{attribute 'enable_dynamic_creation'}
FUNCTION_BLOCK NotificationIterator IMPLEMENTS Iterator
VAR
	pNotificationList 	: ARRAY[0..Param.MAX_ITERABLE_ITEMS] OF POINTER TO Notification;
	//pNotification 		: POINTER TO Notification; 
	nPosition 			: INT := 0;
END_VAR

METHOD current : Object
VAR
	pNotification 		: POINTER TO Notification; 
END_VAR
pNotification := THIS^.pNotificationList[nPosition];
current := pNotification^;
END_METHOD

METHOD FB_init : BOOL
VAR_INPUT
	bInitRetains : BOOL; // if TRUE, the retain variables are initialized (warm start / cold start)
	bInCopyCode : BOOL;  // if TRUE, the instance afterwards gets moved into the copy code (online change)
	pNotificationList : ARRAY[0..Param.MAX_ITERABLE_ITEMS] OF POINTER TO Notification;
END_VAR
This^.pNotificationList := pNotificationList;
END_METHOD

METHOD hasNext : BOOL
IF (THIS^.pNotificationList[nPosition + 1] <> 16#0000) THEN
	hasNext := TRUE;
ELSE
	hasNext := FALSE;	
END_IF
END_METHOD

METHOD next : Object
VAR
	pNotification 		: POINTER TO Notification; 
END_VAR
THIS^.nPosition := THIS^.nPosition + 1;

pNotification := THIS^.pNotificationList[nPosition];
next := pNotification^;
END_METHOD

PROPERTY Position : INT
GET
Position := nPosition;
END_GET
END_PROPERTY

METHOD reset : BOOL
reset := FALSE;

THIS^.nPosition := 0;
reset := TRUE;
END_METHOD

END_FUNCTION_BLOCK

(* stored: Version 1.1.0.1, ProductVersion 3.1.4024.12
   POU NotificationIterator: Id {d6413826-61c3-4c4f-a428-bb95e0e149a0}, SpecialFunc None
   Method current: Id {de0d8d4f-a88b-47fb-ae95-f156b60e189f}
   Method FB_init: Id {74440f01-e5bd-4487-8e42-8c49e9c9c386}
   Method hasNext: Id {0e325456-d50f-42ae-97c1-cc521b11fb76}
   Method next: Id {fe8fab4f-1501-447a-926f-3896c3481b98}
   Property Position: Id {1e16d1d3-ca17-451f-8512-cf2ae4cb9706}
   Get Get: Id {f045d35f-7bb0-475a-bf46-dde5b36582ad}
   Method reset: Id {339a6f97-1a8f-43f4-9ecf-7cf24e122f8f} *)
